{attribute 'strict'}
{attribute 'qualified_only'}
{attribute 'to_string'}
TYPE E_CylFault :
(
	None                  := 0,
    TimeoutExtend         := 1,  // 預期伸出但到位逾時
    TimeoutRetract        := 2,  // 預期縮回但到位逾時
    BothSensorsOn         := 3,  // 原點與末端同時為真（邏輯矛盾/配線錯）
    CoilConflict          := 4,  // 兩線圈同時為真（監測到）
    SensorStuck           := 5   // 感測卡住（可選，見下方邏輯）
);
END_TYPE

(* stored: Version 1.1.0.1, ProductVersion 3.1.4024.15
   EnumerationTextList E_CylFault: Id {685a65f6-221f-4fdc-9178-f7e14cfce148} *)
